// TIA Portal V20 export
TYPE "EmDataBackUp"
// stored: Access Published, Namespace Unit1
   STRUCT
      setPoint : Array[0..10] of "Unit1.posSetpoint";
   END_STRUCT;
END_TYPE
